FUNCTION_BLOCK Compressor
VAR_INPUT
	switch: BOOL;
	
END_VAR
VAR_OUTPUT
END_VAR
VAR
	R_TRIG_0: R_TRIG;
	R_TRIG0: BOOL;
	R_TRIG_1: R_TRIG;
	R_TRIG1: BOOL;
	R_TRIG_2: R_TRIG;
	R_TRIG2: BOOL;
END_VAR


R_TRIG_0(CLK := GVL.GrnBtn, Q=> R_TRIG0);
R_TRIG_1(CLK := GVL.REDBtn, Q=> R_TRIG1);
R_TRIG_2(CLK := GVL.Switch, Q=> R_TRIG2);

IF R_TRIG2 = TRUE THEN
	GVL.Compressor := FALSE;
END_IF


IF switch = FALSE THEN
	GVL.Compressor := TRUE;
ELSE

	IF  R_TRIG0 = TRUE THEN
		GVL.Compressor := TRUE;
	END_IF
	IF  R_TRIG1 = TRUE THEN
		GVL.Compressor := FALSE;
	END_IF 
	
END_IF;

END_FUNCTION_BLOCK

(* stored: Version 1.1.0.1, ProductVersion 3.1.4024.12
   POU Compressor: Id {cc4b9394-775e-43e2-b106-a8314d92dfa9}, SpecialFunc None *)
